(* PLC project Unnamed, Unknown Unnamed 1 *)
(* stored: creationDateTime 2025-03-06T12:52:57, modificationDateTime 2025-03-06T13:12:56 *)

(* Test1 *)
PROGRAM program0

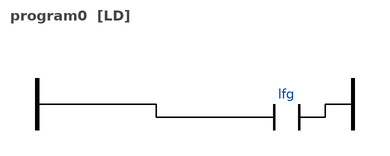
(* LD diagram, written out as Structured Text *)
(* drawn but not wired to any output: lfg *)
END_PROGRAM

CONFIGURATION Config0
  RESOURCE Res0 ON PLC
    TASK task0(INTERVAL := T#20ms, PRIORITY := 0);
    PROGRAM instance0 WITH task0 : program0;
  END_RESOURCE
END_CONFIGURATION
